FUNCTION_BLOCK CS_Recipe
VAR_INPUT
END_VAR
VAR_OUTPUT
END_VAR
VAR
	


 //recipeManCommands: RecipeManCommands;
	result: DWORD;
END_VAR

VAR_IN_OUT
  iRecipe2:    IRecipe;
END_VAR





(*

IF iRecipe2.bCreate THEN
   result:= recipeManCommands.CreateRecipe(RecipeDefinitionName:='Recipes' , RecipeName:='SJ_Rec' );
   iRecipe2.bCreate:=FALSE;
END_IF

IF iRecipe2.bSave THEN
    result:= recipeManCommands.ReadAndSaveRecipeAs(RecipeDefinitionName:='Recipes' , RecipeName:='SJ_Rec' , FileName:='C:\P2Data\P2Par');
    iRecipe2.bSave:=FALSE;
END_IF

IF iRecipe2.bLoad THEN
	result:= RecipeManCommands.LoadFromAndWriteRecipe(RecipeDefinitionName:='Recipes' , RecipeName:='SJ_Rec' , FileName:='C:\P2Data\P2Par');
    iRecipe2.bLoad:=FALSE;
END_IF

*)

END_FUNCTION_BLOCK

(* stored: Version 1.1.0.1, ProductVersion 3.1.4024.9
   POU CS_Recipe: Id {7f8d63df-18b7-43f7-9754-a56b53364943}, SpecialFunc None *)
